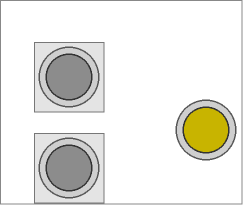
VISUALIZATION Visualization  // 243x205
    Lamp1 (171,95 70x70), variable: MAIN.lamppu, style: Lamp-Lamp1-Yellow
    PushSwitch (34,42 70x70), variable: MAIN.start, behaviour: TAP, style: Switch-PushSwitch-Gray
    PushSwitch (34,133 70x70), variable: MAIN.stop, behaviour: TAP, style: Switch-PushSwitch-Gray
END_VISUALIZATION

(* stored: Version 1.1.0.1, ProductVersion 3.1.4024.0
   Visu Visualization: Id {0f7b54d3-7c47-4008-8132-ad16115b77c1} *)
